(* IEC 61131-3 sources: RL_MAR/experiments/comparison/autoplc/results/qwen3.5-9b_20260511_180311/hf_1, 1 file *)

(* ---- hf_1_1.st ---- *)
FUNCTION_BLOCK StackMin
VAR_INPUT
push : BOOL;
pop : BOOL;
reset : BOOL;
END_VAR
VAR_OUTPUT
error : BOOL;
status : WORD;
END_VAR
VAR_IN_OUT
item : INT;
stack : ARRAY[0..3] OF INT;
END_VAR
VAR
top : INT := -1;
i : INT;
minIndex : INT;
minValue : INT;
END_VAR

error := FALSE;
status := 16#0000;

IF reset THEN
    top := -1;
ELSIF push THEN
    IF top = 3 THEN
        error := TRUE;
        status := 16#8A04;
    ELSE
        top := top + 1;
        stack[top] := item;
        error := FALSE;
        status := 16#0000;
    END_IF;
ELSIF pop THEN
    IF top = -1 THEN
        error := TRUE;
        status := 16#8A05;
    ELSE
        minValue := stack[0];
        minIndex := 0;

        FOR i := 1 TO top DO
            IF stack[i] < minValue THEN
                minValue := stack[i];
                minIndex := i;
            END_IF;
        END_FOR;

        item := minValue;

        FOR i := minIndex TO top - 1 DO
            stack[i] := stack[i + 1];
        END_FOR;

        top := top - 1;
        error := FALSE;
        status := 16#0000;
    END_IF;
END_IF;

END_FUNCTION_BLOCK
